// TIA Portal V17 export
// export: Created 2025-03-07T09:19:34.3940223Z, ExportSetting WithDefaults, DisplayName Totally Integrated Automation Portal, DisplayVersion V17 Update 8, DisplayName TIA Portal Openness, DisplayVersion V17 Update 8, DisplayName TIA Portal Version Control Interface, DisplayVersion V17, DisplayName SINAMICS Startdrive Advanced, DisplayVersion V17 SP2, DisplayName SINAMICS Startdrive G110M, G120, G120C, G120D, G120P, G115D, DisplayVersion V17 SP2, DisplayName SINAMICS Startdrive G130, G150, S120, S150, SINAMICS MV, S210, DisplayVersion V17 SP2, DisplayName STEP 7 Professional, DisplayVersion V17 Update 8, DisplayName SINUMERIK ONE STEP 7 Toolbox, DisplayVersion V17 Update 12, DisplayName SINUMERIK 840D sl STEP 7 Toolbox, DisplayVersion V17 Update 12, DisplayName STEP 7 Safety, DisplayVersion V17 Update 6, DisplayName WinCC Advanced, DisplayVersion V17 Update 8
TYPE "LBP_typeModularMcpBaseInput"
TITLE = Modular MCP image / Imagen de MCP modulares / Abbild modulare MCP
// Input image of base signals for modular MCP / Imagen de entrada de señales base de MCP modulares / Eingangsabbild von Basissignalen für modulare MCP
// stored: IsFailsafeCompliant false
   STRUCT
      optionalKey1 : Bool;   // Eingangsabbild n+0 Bit 0; KT-IN1 / input image n+0 bit 0; KT-IN1 / Imagen de entrada n+0 bit 0; KT-IN1
      optionalKey2 : Bool;   // Eingangsabbild n+0 Bit 1; KT-IN2 / input image n+0 bit 1; KT-IN2 / Imagen de entrada n+0 bit 1; KT-IN2
      optionalKey3 : Bool;   // Eingangsabbild n+0 Bit 2; KT-IN3 / input image n+0 bit 2; KT-IN3 / Imagen de entrada n+0 bit 2; KT-IN3
      optionalKey4 : Bool;   // Eingangsabbild n+0 Bit 3; KT-IN4 / input image n+0 bit 3; KT-IN4 / Imagen de entrada n+0 bit 3; KT-IN4
      optionalKey5 : Bool;   // Eingangsabbild n+0 Bit 4; KT-IN5 / input image n+0 bit 4; KT-IN5 / Imagen de entrada n+0 bit 4; KT-IN5
      optionalKey6 : Bool;   // Eingangsabbild n+0 Bit 5; KT-IN6 / input image n+0 bit 5; KT-IN6 / Imagen de entrada n+0 bit 5; KT-IN6
      optionalKey7 : Bool;   // Eingangsabbild n+0 Bit 6; KT-IN7 / input image n+0 bit 6; KT-IN7 / Imagen de entrada n+0 bit 6; KT-IN7
      optionalKey8 : Bool;   // Eingangsabbild n+0 Bit 7; KT-IN8 / input image n+0 bit 7; KT-IN8 / Imagen de entrada n+0 bit 7; KT-IN8
      optionalKey9 : Bool;   // Eingangsabbild n+1 Bit 0; KT-IN9 / input image n+1 bit 0; KT-IN9 / Imagen de entrada n+1 bit 0; KT-IN9
      optionalKey10 : Bool;   // Eingangsabbild n+1 Bit 1; KT-IN10 / input image n+1 bit 1; KT-IN10 / Imagen de entrada n+1 bit 1; KT-IN10
      optionalKey11 : Bool;   // Eingangsabbild n+1 Bit 2; KT-IN11 / input image n+1 bit 2; KT-IN11 / Imagen de entrada n+1 bit 2; KT-IN11
      optionalKey12 : Bool;   // Eingangsabbild n+1 Bit 3; KT-IN12 / input image n+1 bit 3; KT-IN12 / Imagen de entrada n+1 bit 3; KT-IN12
      optionalKey13 : Bool;   // Eingangsabbild n+1 Bit 4; KT-IN13 / input image n+1 bit 4; KT-IN13 / Imagen de entrada n+1 bit 4; KT-IN13
      optionalKey14 : Bool;   // Eingangsabbild n+1 Bit 5; KT-IN14 / input image n+1 bit 5; KT-IN14 / Imagen de entrada n+1 bit 5; KT-IN14
      optionalKey15 : Bool;   // Eingangsabbild n+1 Bit 6; KT-IN15 / input image n+1 bit 6; KT-IN15 / Imagen de entrada n+1 bit 6; KT-IN15
      optionalKey16 : Bool;   // Eingangsabbild n+1 Bit 7; KT-IN16 / input image n+1 bit 7; KT-IN16 / Imagen de entrada n+1 bit 7; KT-IN16
      spindleOvr : USInt;   // Eingangsabbild Byte n+2 / input image byte n+2 / Imagen de entrada byte n+2
      feedrateOvr : USInt;   // Eingangsabbild Byte n+3 / input image byte n+3 / Imagen de entrada byte n+3
      keySwitch0 : Bool;   // Eingangsabbild n+4 Bit 0 / input image n+4 bit 0 / Imagen de entrada n+4 bit 0
      keySwitch1 : Bool;   // Eingangsabbild n+4 Bit 1 / input image n+4 bit 1 / Imagen de entrada n+4 bit 1
      keySwitch2 : Bool;   // Eingangsabbild n+4 Bit 2 / input image n+4 bit 2 / Imagen de entrada n+4 bit 2
      keySwitch3 : Bool;   // Eingangsabbild n+4 Bit 3 / input image n+4 bit 3 / Imagen de entrada n+4 bit 3
      reserved44 : Bool;
      reserved45 : Bool;
      reserved46 : Bool;
      reserved47 : Bool;
      reserved50 : Bool;
      reserved51 : Bool;
      reserved52 : Bool;
      reserved53 : Bool;
      reserved54 : Bool;
      reserved55 : Bool;
      reserved56 : Bool;
      reserved57 : Bool;
   END_STRUCT;
END_TYPE
